// TIA Portal V19 export
FUNCTION_BLOCK "F_Zone15_FB"   // FB190, F_LAD
TITLE = SAFETY ZONE 11 - AREA 02 (PROFILATRICE)
// -
// stored: Access Published
   VAR
      D16 : "Door_FB";
      D18 : "Door_FB";
      FNS : "ForceNormalStop";
      F_Sinamics_AccRolls1 { ExternalAccessible := 'False'; ExternalVisible := 'False'; ExternalWritable := 'False'} : "FDevice_Sinamics_FB";
      F_Sinamics_AccRolls2 { ExternalAccessible := 'False'; ExternalVisible := 'False'; ExternalWritable := 'False'} : "FDevice_Sinamics_FB";
      F_Sinamics_AccRolls3 { ExternalAccessible := 'False'; ExternalVisible := 'False'; ExternalWritable := 'False'} : "FDevice_Sinamics_FB";
   END_VAR
   VAR_TEMP
      DoorNormalStop : Bool;
      DoorSafeStop : Bool;
      Door_Ok : Bool;
   END_VAR
   VAR CONSTANT
      ACCROLLS_S120_STOPPING_TIME : Time := T#1s;
   END_VAR
BEGIN

REGION Network 1: < < < < < < < < < < DOOR > > > > > > > > > >
END_REGION

REGION Network 2: Zone Entry enable
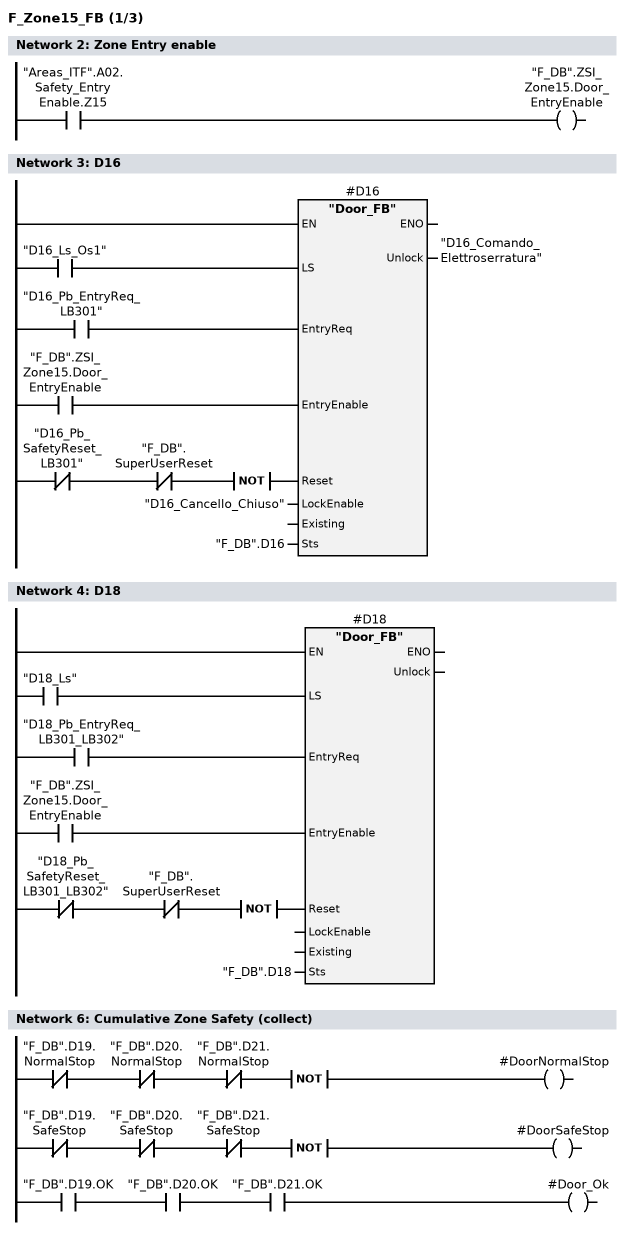
   RUNG wire#powerrail
      Contact( "Areas_ITF".A02.Safety_EntryEnable.Z15 )
      Coil( "F_DB".ZSI_Zone15.Door_EntryEnable )
   END_RUNG
   // the same network as SCL:
   "F_DB".ZSI_Zone15.Door_EntryEnable := "Areas_ITF".A02.Safety_EntryEnable.Z15;
END_REGION

REGION Network 3: D16
   RUNG wire#powerrail
      #D16(LS := wire#w1, EntryReq := wire#w2, EntryEnable := wire#w3, Reset := wire#w4, LockEnable := "D16_Cancello_Chiuso", Existing :=, Sts := "F_DB".D16, Unlock => "D16_Comando_Elettroserratura")
   END_RUNG
   RUNG wire#powerrail
      Contact( "D16_Ls_Os1" )
   END_RUNG wire#w1
   RUNG wire#powerrail
      Contact( "D16_Pb_EntryReq_LB301" )
   END_RUNG wire#w2
   RUNG wire#powerrail
      Contact( "F_DB".ZSI_Zone15.Door_EntryEnable )
   END_RUNG wire#w3
   RUNG wire#powerrail
      I_Contact( "D16_Pb_SafetyReset_LB301" )
      I_Contact( "F_DB".SuperUserReset )
      Not()
   END_RUNG wire#w4
   // the same network as SCL:
   #D16(LS := "D16_Ls_Os1",   // "Door_FB"
        EntryReq := "D16_Pb_EntryReq_LB301",
        EntryEnable := "F_DB".ZSI_Zone15.Door_EntryEnable,
        Reset := NOT (NOT "D16_Pb_SafetyReset_LB301" AND NOT "F_DB".SuperUserReset),
        LockEnable := "D16_Cancello_Chiuso",
        Sts := "F_DB".D16,
        Unlock => "D16_Comando_Elettroserratura");
END_REGION

REGION Network 4: D18
   RUNG wire#powerrail
      #D18(LS := wire#w1, EntryReq := wire#w2, EntryEnable := wire#w3, Reset := wire#w4, LockEnable :=, Existing :=, Sts := "F_DB".D18, Unlock =>)
   END_RUNG
   RUNG wire#powerrail
      Contact( "D18_Ls" )
   END_RUNG wire#w1
   RUNG wire#powerrail
      Contact( "D18_Pb_EntryReq_LB301_LB302" )
   END_RUNG wire#w2
   RUNG wire#powerrail
      Contact( "F_DB".ZSI_Zone15.Door_EntryEnable )
   END_RUNG wire#w3
   RUNG wire#powerrail
      I_Contact( "D18_Pb_SafetyReset_LB301_LB302" )
      I_Contact( "F_DB".SuperUserReset )
      Not()
   END_RUNG wire#w4
   // the same network as SCL:
   #D18(LS := "D18_Ls",   // "Door_FB"
        EntryReq := "D18_Pb_EntryReq_LB301_LB302",
        EntryEnable := "F_DB".ZSI_Zone15.Door_EntryEnable,
        Reset := NOT (NOT "D18_Pb_SafetyReset_LB301_LB302" AND NOT "F_DB".SuperUserReset),
        Sts := "F_DB".D18);
END_REGION

REGION Network 5: < < < < < < < < < < ZONE SAFETY INTERFACE > > > > > > > > > >
END_REGION

REGION Network 6: Cumulative Zone Safety (collect)
   RUNG wire#powerrail
      I_Contact( "F_DB".D19.NormalStop )
      I_Contact( "F_DB".D20.NormalStop )
      I_Contact( "F_DB".D21.NormalStop )
      Not()
      Coil( #DoorNormalStop )
   END_RUNG
   RUNG wire#powerrail
      I_Contact( "F_DB".D19.SafeStop )
      I_Contact( "F_DB".D20.SafeStop )
      I_Contact( "F_DB".D21.SafeStop )
      Not()
      Coil( #DoorSafeStop )
   END_RUNG
   RUNG wire#powerrail
      Contact( "F_DB".D19.OK )
      Contact( "F_DB".D20.OK )
      Contact( "F_DB".D21.OK )
      Coil( #Door_Ok )
   END_RUNG
   // the same network as SCL:
   #DoorNormalStop := NOT (NOT "F_DB".D19.NormalStop AND NOT "F_DB".D20.NormalStop AND NOT "F_DB".D21.NormalStop);
   #DoorSafeStop := NOT (NOT "F_DB".D19.SafeStop AND NOT "F_DB".D20.SafeStop AND NOT "F_DB".D21.SafeStop);
   #Door_Ok := "F_DB".D19.OK AND "F_DB".D20.OK AND "F_DB".D21.OK;
END_REGION

REGION Network 7: Zone must stay in Normal Stop During Restart
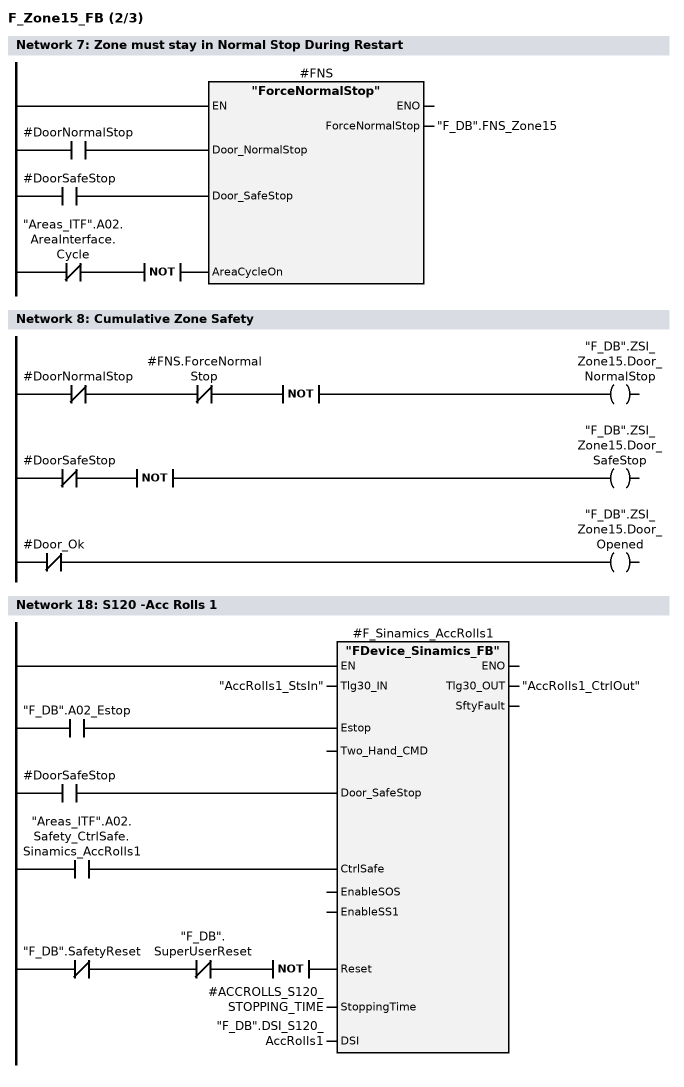
   RUNG wire#powerrail
      #FNS(Door_NormalStop := wire#w1, Door_SafeStop := wire#w2, AreaCycleOn := wire#w3, ForceNormalStop => "F_DB".FNS_Zone15)
   END_RUNG
   RUNG wire#powerrail
      Contact( #DoorNormalStop )
   END_RUNG wire#w1
   RUNG wire#powerrail
      Contact( #DoorSafeStop )
   END_RUNG wire#w2
   RUNG wire#powerrail
      I_Contact( "Areas_ITF".A02.AreaInterface.Cycle )
      Not()
   END_RUNG wire#w3
   // the same network as SCL:
   #FNS(Door_NormalStop := #DoorNormalStop,   // "ForceNormalStop"
        Door_SafeStop := #DoorSafeStop,
        AreaCycleOn := NOT (NOT "Areas_ITF".A02.AreaInterface.Cycle),
        ForceNormalStop => "F_DB".FNS_Zone15);
END_REGION

REGION Network 8: Cumulative Zone Safety
   RUNG wire#powerrail
      I_Contact( #DoorNormalStop )
      I_Contact( #FNS.ForceNormalStop )
      Not()
      Coil( "F_DB".ZSI_Zone15.Door_NormalStop )
   END_RUNG
   RUNG wire#powerrail
      I_Contact( #DoorSafeStop )
      Not()
      Coil( "F_DB".ZSI_Zone15.Door_SafeStop )
   END_RUNG
   RUNG wire#powerrail
      I_Contact( #Door_Ok )
      Coil( "F_DB".ZSI_Zone15.Door_Opened )
   END_RUNG
   // the same network as SCL:
   "F_DB".ZSI_Zone15.Door_NormalStop := NOT (NOT #DoorNormalStop AND NOT #FNS.ForceNormalStop);
   "F_DB".ZSI_Zone15.Door_SafeStop := NOT (NOT #DoorSafeStop);
   "F_DB".ZSI_Zone15.Door_Opened := NOT #Door_Ok;
END_REGION

REGION Network 9: >
END_REGION

REGION Network 10: >
END_REGION

REGION Network 11: < < < < < < < < < < DEVICES SAFETY VALVES > > > > > > > > > >
END_REGION

REGION Network 12: >
END_REGION

REGION Network 13: >
END_REGION

REGION Network 14: < < < < < < < < < < DEVICES CONTACTORS > > > > > > > > > >
END_REGION

REGION Network 15: >
END_REGION

REGION Network 16: >
END_REGION

REGION Network 17: < < < < < < < < < < DEVICES S120 > > > > > > > > > >
END_REGION

REGION Network 18: S120 -Acc Rolls 1
   RUNG wire#powerrail
      #F_Sinamics_AccRolls1(Estop := wire#w1, Door_SafeStop := wire#w2, CtrlSafe := wire#w3, Reset := wire#w4, Tlg30_IN := "AccRolls1_StsIn", Two_Hand_CMD :=, EnableSOS :=, EnableSS1 :=, StoppingTime := #ACCROLLS_S120_STOPPING_TIME, DSI := "F_DB".DSI_S120_AccRolls1, Tlg30_OUT => "AccRolls1_CtrlOut", SftyFault =>)
   END_RUNG
   RUNG wire#powerrail
      Contact( "F_DB".A02_Estop )
   END_RUNG wire#w1
   RUNG wire#powerrail
      Contact( #DoorSafeStop )
   END_RUNG wire#w2
   RUNG wire#powerrail
      Contact( "Areas_ITF".A02.Safety_CtrlSafe.Sinamics_AccRolls1 )
   END_RUNG wire#w3
   RUNG wire#powerrail
      I_Contact( "F_DB".SafetyReset )
      I_Contact( "F_DB".SuperUserReset )
      Not()
   END_RUNG wire#w4
   // the same network as SCL:
   #F_Sinamics_AccRolls1(Tlg30_IN := "AccRolls1_StsIn",   // "FDevice_Sinamics_FB"
                         Estop := "F_DB".A02_Estop,
                         Door_SafeStop := #DoorSafeStop,
                         CtrlSafe := "Areas_ITF".A02.Safety_CtrlSafe.Sinamics_AccRolls1,
                         Reset := NOT (NOT "F_DB".SafetyReset AND NOT "F_DB".SuperUserReset),
                         StoppingTime := #ACCROLLS_S120_STOPPING_TIME,
                         DSI := "F_DB".DSI_S120_AccRolls1,
                         Tlg30_OUT => "AccRolls1_CtrlOut");
END_REGION

REGION Network 19: S120 -Acc Rolls 2
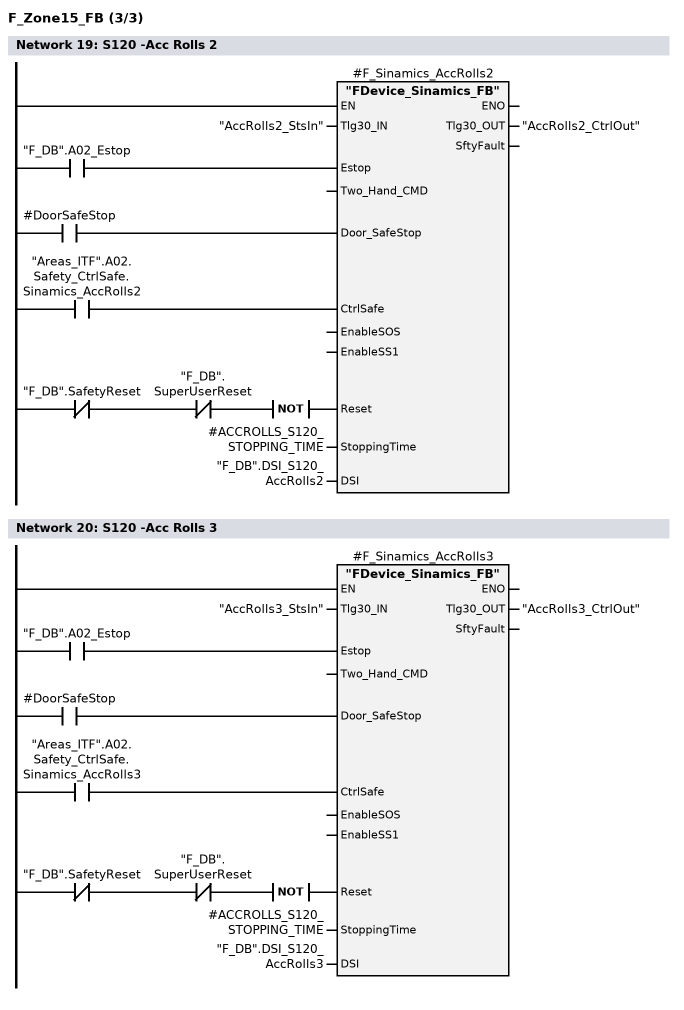
   RUNG wire#powerrail
      #F_Sinamics_AccRolls2(Estop := wire#w1, Door_SafeStop := wire#w2, CtrlSafe := wire#w3, Reset := wire#w4, Tlg30_IN := "AccRolls2_StsIn", Two_Hand_CMD :=, EnableSOS :=, EnableSS1 :=, StoppingTime := #ACCROLLS_S120_STOPPING_TIME, DSI := "F_DB".DSI_S120_AccRolls2, Tlg30_OUT => "AccRolls2_CtrlOut", SftyFault =>)
   END_RUNG
   RUNG wire#powerrail
      Contact( "F_DB".A02_Estop )
   END_RUNG wire#w1
   RUNG wire#powerrail
      Contact( #DoorSafeStop )
   END_RUNG wire#w2
   RUNG wire#powerrail
      Contact( "Areas_ITF".A02.Safety_CtrlSafe.Sinamics_AccRolls2 )
   END_RUNG wire#w3
   RUNG wire#powerrail
      I_Contact( "F_DB".SafetyReset )
      I_Contact( "F_DB".SuperUserReset )
      Not()
   END_RUNG wire#w4
   // the same network as SCL:
   #F_Sinamics_AccRolls2(Tlg30_IN := "AccRolls2_StsIn",   // "FDevice_Sinamics_FB"
                         Estop := "F_DB".A02_Estop,
                         Door_SafeStop := #DoorSafeStop,
                         CtrlSafe := "Areas_ITF".A02.Safety_CtrlSafe.Sinamics_AccRolls2,
                         Reset := NOT (NOT "F_DB".SafetyReset AND NOT "F_DB".SuperUserReset),
                         StoppingTime := #ACCROLLS_S120_STOPPING_TIME,
                         DSI := "F_DB".DSI_S120_AccRolls2,
                         Tlg30_OUT => "AccRolls2_CtrlOut");
END_REGION

REGION Network 20: S120 -Acc Rolls 3
   RUNG wire#powerrail
      #F_Sinamics_AccRolls3(Estop := wire#w1, Door_SafeStop := wire#w2, CtrlSafe := wire#w3, Reset := wire#w4, Tlg30_IN := "AccRolls3_StsIn", Two_Hand_CMD :=, EnableSOS :=, EnableSS1 :=, StoppingTime := #ACCROLLS_S120_STOPPING_TIME, DSI := "F_DB".DSI_S120_AccRolls3, Tlg30_OUT => "AccRolls3_CtrlOut", SftyFault =>)
   END_RUNG
   RUNG wire#powerrail
      Contact( "F_DB".A02_Estop )
   END_RUNG wire#w1
   RUNG wire#powerrail
      Contact( #DoorSafeStop )
   END_RUNG wire#w2
   RUNG wire#powerrail
      Contact( "Areas_ITF".A02.Safety_CtrlSafe.Sinamics_AccRolls3 )
   END_RUNG wire#w3
   RUNG wire#powerrail
      I_Contact( "F_DB".SafetyReset )
      I_Contact( "F_DB".SuperUserReset )
      Not()
   END_RUNG wire#w4
   // the same network as SCL:
   #F_Sinamics_AccRolls3(Tlg30_IN := "AccRolls3_StsIn",   // "FDevice_Sinamics_FB"
                         Estop := "F_DB".A02_Estop,
                         Door_SafeStop := #DoorSafeStop,
                         CtrlSafe := "Areas_ITF".A02.Safety_CtrlSafe.Sinamics_AccRolls3,
                         Reset := NOT (NOT "F_DB".SafetyReset AND NOT "F_DB".SuperUserReset),
                         StoppingTime := #ACCROLLS_S120_STOPPING_TIME,
                         DSI := "F_DB".DSI_S120_AccRolls3,
                         Tlg30_OUT => "AccRolls3_CtrlOut");
END_REGION

REGION Network 21: >
END_REGION

REGION Network 22: >
END_REGION
END_FUNCTION_BLOCK
